Fanuc TP program (LS listing): UP021.LS

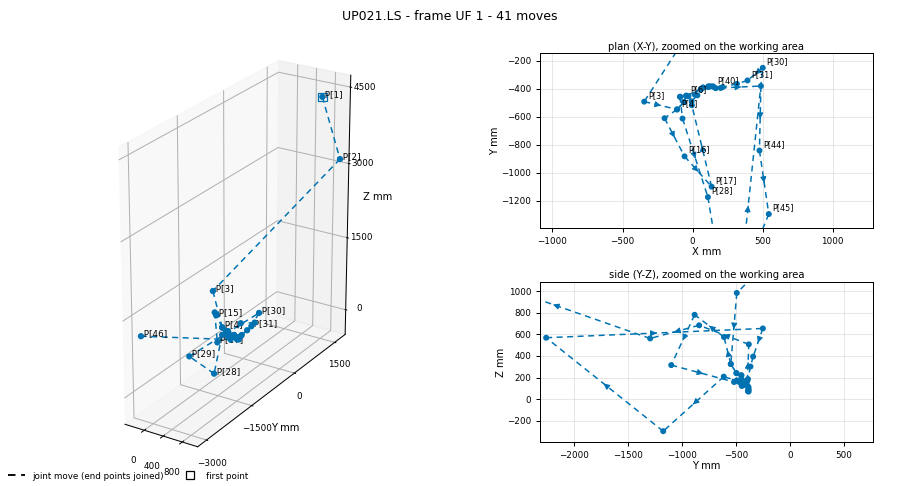
[picture p0: tool path of UP021.LS in frame UF 1, 41 of 46 moves have a stored position in this frame; points joined in program order, loops and branches not executed]
/PROG  UP021
/ATTR
OWNER		= GME;
COMMENT		= "Soldar en ST1120";
PROG_SIZE	= 17280;
CREATE		= DATE 96-06-10  TIME 20:13:44;
MODIFIED	= DATE 23-11-12  TIME 10:55:54;
FILE_NAME	= UP021;
VERSION		= 0;
LINE_COUNT	= 61;
MEMORY_SIZE	= 34620;
PROTECT		= READ_WRITE;
TCD:  STACK_SIZE	= 500,
      TASK_PRIORITY	= 50,
      TIME_SLICE	= 0,
      BUSY_LAMP_OFF	= 0,
      ABORT_REQUEST	= 0,
      PAUSE_REQUEST	= 0;
DEFAULT_GROUP	= 1,1,1,1,*;
CONTROL_CODE	= 00000000 00000000;
/APPL
/MN
   1:  UFRAME_NUM=1 ;
   2:  UTOOL_NUM=1 ;
   3:  PAYLOAD[1] ;
   4:J P[1] 100% CNT0 ACC100 TB    0.00sec,P-SPS    ;
      1:  TC_ONLINE (ON) ;
      2:  DO[23:Bloquear Rejas de Seg.]=OFF ;
      3:  TIMER[3]=RESET ;
      4:  TIMER[3]=START ;
      5:  CALL MAKRO050    ;
      6:  !Lib. de Herramientas ;
      7:  DO[80:PL>Cortina Seg.]=ON ;
      8:  DO[79:PL>1120 Herramienta]=ON ;
      9:  DO[78:Ctrl.1120 Cil.]=OFF ;
     10:  DO[77:Pos.Tomar 1120]=OFF ;
     11:  DO[76:PL>1125 Dep�sito]=ON ;
     12:  DO[74:Pos.Dejar 1125]=OFF ;
     13:  !Lib. de Anticolisiones ;
     14:  DO[41:Blq>1130R01(1)]=ON ;
     15:  DO[42:Blq>1130R01(2)]=ON ;
     16:  !Apagar Pos. Base ;
     17:  DO[15:PF0 Robot (Punto Cero)]=OFF ;
     18:  !Robot en Trayectoria ;
     19:  DO[16:SAK Robot (En camino)]=ON ;
     20:  WAIT (DI[80:Cortina Abajo] AND DI[79:1120 Soldar])    ;
     21:  DO[80:PL>Cortina Seg.]=OFF ;
     22:  DO[79:PL>1120 Herramienta]=OFF ;
     23:  WAIT (DI[23:Sin Sol.Acceso])    ;
     24:  DO[23:Bloquear Rejas de Seg.]=ON ;
     25:  TC_ONLINE (DI[80:Cortina Abajo] AND DI[79:1120 Soldar] AND M[2:Garra Vacia] AND M[30:Seg. de M�quina] AND M[31:Gpo.Suj. 1 Abierto] AND M[33:Gpo.Suj. 2 Abierto] AND M[95:Seguridad SP1] AND M[102:Seguridad SP2] AND
       :  M[103:KS2 En Reposo]) ;
       ------ ;
   5:J P[2] 100% CNT100 ACC100 TB   0.00sec,P-SPS    ;
      1:  TC_ONLINE (DI[80:Cortina Abajo] AND DI[79:1120 Soldar] AND M[2:Garra Vacia] AND M[30:Seg. de M�quina] AND M[31:Gpo.Suj. 1 Abierto] AND M[33:Gpo.Suj. 2 Abierto] AND M[95:Seguridad SP1] AND M[102:Seguridad SP2] AND
       :  M[103:KS2 En Reposo]) ;
       ------ ;
   6:J P[3] 100% CNT100 ACC100 TB   0.00sec,P-SPS    ;
      1:  TC_ONLINE (DI[80:Cortina Abajo] AND DI[79:1120 Soldar] AND M[2:Garra Vacia] AND M[30:Seg. de M�quina] AND M[31:Gpo.Suj. 1 Abierto] AND M[33:Gpo.Suj. 2 Abierto] AND M[95:Seguridad SP1] AND M[102:Seguridad SP2] AND
       :  M[103:KS2 En Reposo]) ;
       ------ ;
   7:J P[4] 100% CNT100 ACC100 TB   0.00sec,P-SPS    ;
      1:  TC_ONLINE (DI[80:Cortina Abajo] AND DI[79:1120 Soldar] AND M[2:Garra Vacia] AND M[30:Seg. de M�quina] AND M[31:Gpo.Suj. 1 Abierto] AND M[33:Gpo.Suj. 2 Abierto] AND M[95:Seguridad SP1] AND M[102:Seguridad SP2] AND
       :  M[103:KS2 En Reposo]) ;
       ------ ;
   8:J P[5] 100% CNT100 ACC100 TB   0.00sec,P-SPS    ;
      1:  TC_ONLINE (DI[80:Cortina Abajo] AND DI[79:1120 Soldar] AND M[2:Garra Vacia] AND M[30:Seg. de M�quina] AND M[31:Gpo.Suj. 1 Abierto] AND M[33:Gpo.Suj. 2 Abierto] AND M[95:Seguridad SP1] AND M[102:Seguridad SP2] AND
       :  M[103:KS2 En Reposo]) ;
       ------ ;
   9:J P[6] 100% CNT100 ACC100 TB   0.00sec,P-SPS    ;
      1:  TC_ONLINE (DI[80:Cortina Abajo] AND DI[79:1120 Soldar] AND M[2:Garra Vacia] AND M[30:Seg. de M�quina] AND M[31:Gpo.Suj. 1 Abierto] AND M[33:Gpo.Suj. 2 Abierto] AND M[95:Seguridad SP1] AND M[102:Seguridad SP2] AND
       :  M[103:KS2 En Reposo]) ;
       ------ ;
  10:J P[7] 100% CNT25 ACC100 TB   0.00sec,P-SPS    ;
      1:  TC_ONLINE (DI[80:Cortina Abajo] AND DI[79:1120 Soldar] AND M[2:Garra Vacia] AND M[30:Seg. de M�quina] AND M[31:Gpo.Suj. 1 Abierto] AND M[33:Gpo.Suj. 2 Abierto] AND M[95:Seguridad SP1] AND M[102:Seguridad SP2] AND
       :  M[103:KS2 En Reposo]) ;
       ------ ;
  11:J P[8] 100% CNT100 ACC100 TB   0.00sec,P-SPS    ;
      1:  TC_ONLINE (DI[80:Cortina Abajo] AND DI[79:1120 Soldar] AND M[2:Garra Vacia] AND M[30:Seg. de M�quina] AND M[31:Gpo.Suj. 1 Abierto] AND M[33:Gpo.Suj. 2 Abierto] AND M[95:Seguridad SP1] AND M[102:Seguridad SP2] AND
       :  M[103:KS2 En Reposo]) ;
       ------ ;
  12:  !5qa802035b_027_abps0002_L ;
  13:  !Punto de Sol. No. 10001 ;
  14:J P[9] 100% CNT0 ACC100 TB    .10sec,P-SPS Tool_Offset,PR[11] Offset,PR[12]    ;
      1:  TC_ONLINE (ON) ;
      2:  DO[23:Bloquear Rejas de Seg.]=OFF ;
      3:  WAIT (!DI[16:Paro Correcciones] AND DI[23:Sin Sol.Acceso])    ;
      4:  CALL VW_USER(Basic1,EZSP,Nr1,ProgNr=99, , ,S-Punkt=10001,Fzg_Typ=7,EIN/AUS=ON) ;
      5:  GO[2:SP1 Compensaci�n]=(R[197]) ;
      6:  WAIT (!DI[129:SZ1 Sin Fuerza] OR DI[26:Conf.Repetir])    ;
      7:  CALL MAKRO080    ;
      8:  WAIT (DI[23:Sin Sol.Acceso])    ;
      9:  DO[23:Bloquear Rejas de Seg.]=ON ;
     10:  TC_ONLINE (DI[80:Cortina Abajo] AND DI[79:1120 Soldar] AND M[2:Garra Vacia] AND M[30:Seg. de M�quina] AND M[31:Gpo.Suj. 1 Abierto] AND M[33:Gpo.Suj. 2 Abierto] AND M[95:Seguridad SP1] AND M[102:Seguridad SP2] AND
       :  M[103:KS2 En Reposo]) ;
       ------ ;
  15:J P[10] 100% CNT100 ACC100 TB   0.00sec,P-SPS    ;
      1:  TC_ONLINE (DI[80:Cortina Abajo] AND DI[79:1120 Soldar] AND M[2:Garra Vacia] AND M[30:Seg. de M�quina] AND M[31:Gpo.Suj. 1 Abierto] AND M[33:Gpo.Suj. 2 Abierto] AND M[95:Seguridad SP1] AND M[102:Seguridad SP2] AND
       :  M[103:KS2 En Reposo]) ;
       ------ ;
  16:J P[11] 100% CNT25 ACC100 TB   0.00sec,P-SPS    ;
      1:  TC_ONLINE (DI[80:Cortina Abajo] AND DI[79:1120 Soldar] AND M[2:Garra Vacia] AND M[30:Seg. de M�quina] AND M[31:Gpo.Suj. 1 Abierto] AND M[33:Gpo.Suj. 2 Abierto] AND M[95:Seguridad SP1] AND M[102:Seguridad SP2] AND
       :  M[103:KS2 En Reposo]) ;
       ------ ;
  17:J P[12] 100% CNT100 ACC100 TB   0.00sec,P-SPS    ;
      1:  TC_ONLINE (DI[80:Cortina Abajo] AND DI[79:1120 Soldar] AND M[2:Garra Vacia] AND M[30:Seg. de M�quina] AND M[31:Gpo.Suj. 1 Abierto] AND M[33:Gpo.Suj. 2 Abierto] AND M[95:Seguridad SP1] AND M[102:Seguridad SP2] AND
       :  M[103:KS2 En Reposo]) ;
       ------ ;
  18:J P[13] 100% CNT100 ACC100 TB   0.00sec,P-SPS    ;
      1:  TC_ONLINE (DI[80:Cortina Abajo] AND DI[79:1120 Soldar] AND M[2:Garra Vacia] AND M[30:Seg. de M�quina] AND M[31:Gpo.Suj. 1 Abierto] AND M[33:Gpo.Suj. 2 Abierto] AND M[95:Seguridad SP1] AND M[102:Seguridad SP2] AND
       :  M[103:KS2 En Reposo]) ;
       ------ ;
  19:J P[14] 100% CNT100 ACC100 TB   0.00sec,P-SPS    ;
      1:  TC_ONLINE (DI[80:Cortina Abajo] AND DI[79:1120 Soldar] AND M[2:Garra Vacia] AND M[30:Seg. de M�quina] AND M[31:Gpo.Suj. 1 Abierto] AND M[33:Gpo.Suj. 2 Abierto] AND M[95:Seguridad SP1] AND M[102:Seguridad SP2] AND
       :  M[103:KS2 En Reposo]) ;
       ------ ;
  20:J P[15] 100% CNT100 ACC100 TB   0.00sec,P-SPS    ;
      1:  TC_ONLINE (DI[80:Cortina Abajo] AND DI[79:1120 Soldar] AND M[2:Garra Vacia] AND M[30:Seg. de M�quina] AND M[31:Gpo.Suj. 1 Abierto] AND M[33:Gpo.Suj. 2 Abierto] AND M[95:Seguridad SP1] AND M[102:Seguridad SP2] AND
       :  M[103:KS2 En Reposo]) ;
       ------ ;
  21:J P[16] 100% CNT100 ACC100 TB   0.00sec,P-SPS    ;
      1:  TC_ONLINE (DI[80:Cortina Abajo] AND DI[79:1120 Soldar] AND M[2:Garra Vacia] AND M[30:Seg. de M�quina] AND M[31:Gpo.Suj. 1 Abierto] AND M[33:Gpo.Suj. 2 Abierto] AND M[95:Seguridad SP1] AND M[102:Seguridad SP2] AND
       :  M[103:KS2 En Reposo]) ;
       ------ ;
  22:J P[17] 100% CNT100 ACC100 TB   0.00sec,P-SPS    ;
      1:  TC_ONLINE (DI[80:Cortina Abajo] AND DI[79:1120 Soldar] AND M[2:Garra Vacia] AND M[30:Seg. de M�quina] AND M[31:Gpo.Suj. 1 Abierto] AND M[33:Gpo.Suj. 2 Abierto] AND M[95:Seguridad SP1] AND M[102:Seguridad SP2] AND
       :  M[103:KS2 En Reposo]) ;
       ------ ;
  23:J P[18] 100% CNT100 ACC100 TB   0.00sec,P-SPS    ;
      1:  TC_ONLINE (DI[80:Cortina Abajo] AND DI[79:1120 Soldar] AND M[2:Garra Vacia] AND M[30:Seg. de M�quina] AND M[31:Gpo.Suj. 1 Abierto] AND M[33:Gpo.Suj. 2 Abierto] AND M[95:Seguridad SP1] AND M[102:Seguridad SP2] AND
       :  M[103:KS2 En Reposo]) ;
       ------ ;
  24:J P[19] 100% CNT100 ACC100 TB   0.00sec,P-SPS    ;
      1:  TC_ONLINE (DI[80:Cortina Abajo] AND DI[79:1120 Soldar] AND M[2:Garra Vacia] AND M[30:Seg. de M�quina] AND M[31:Gpo.Suj. 1 Abierto] AND M[33:Gpo.Suj. 2 Abierto] AND M[95:Seguridad SP1] AND M[102:Seguridad SP2] AND
       :  M[103:KS2 En Reposo]) ;
       ------ ;
  25:  !5qa802035b_027_abps0005_L ;
  26:  !Punto de Sol. No. 10002 ;
  27:J P[20] 100% CNT0 ACC100 TB    .10sec,P-SPS Tool_Offset,PR[11] Offset,PR[12]    ;
      1:  TC_ONLINE (ON) ;
      2:  DO[23:Bloquear Rejas de Seg.]=OFF ;
      3:  WAIT (!DI[16:Paro Correcciones] AND DI[23:Sin Sol.Acceso])    ;
      4:  CALL VW_USER(Basic1,EZSP,Nr1,ProgNr=99, , ,S-Punkt=10002,Fzg_Typ=7,EIN/AUS=ON) ;
      5:  GO[2:SP1 Compensaci�n]=(R[197]+1) ;
      6:  WAIT (!DI[129:SZ1 Sin Fuerza] OR DI[26:Conf.Repetir])    ;
      7:  CALL MAKRO080    ;
      8:  WAIT (DI[23:Sin Sol.Acceso])    ;
      9:  DO[23:Bloquear Rejas de Seg.]=ON ;
     10:  TC_ONLINE (DI[80:Cortina Abajo] AND DI[79:1120 Soldar] AND M[2:Garra Vacia] AND M[30:Seg. de M�quina] AND M[31:Gpo.Suj. 1 Abierto] AND M[33:Gpo.Suj. 2 Abierto] AND M[95:Seguridad SP1] AND M[102:Seguridad SP2] AND
       :  M[103:KS2 En Reposo]) ;
       ------ ;
  28:J P[21] 100% CNT100 ACC100 TB   0.00sec,P-SPS    ;
      1:  TC_ONLINE (DI[80:Cortina Abajo] AND DI[79:1120 Soldar] AND M[2:Garra Vacia] AND M[30:Seg. de M�quina] AND M[31:Gpo.Suj. 1 Abierto] AND M[33:Gpo.Suj. 2 Abierto] AND M[95:Seguridad SP1] AND M[102:Seguridad SP2] AND
       :  M[103:KS2 En Reposo]) ;
       ------ ;
  29:J P[22] 100% CNT100 ACC100 TB   0.00sec,P-SPS    ;
      1:  TC_ONLINE (DI[80:Cortina Abajo] AND DI[79:1120 Soldar] AND M[2:Garra Vacia] AND M[30:Seg. de M�quina] AND M[31:Gpo.Suj. 1 Abierto] AND M[33:Gpo.Suj. 2 Abierto] AND M[95:Seguridad SP1] AND M[102:Seguridad SP2] AND
       :  M[103:KS2 En Reposo]) ;
       ------ ;
  30:J P[23] 100% CNT100 ACC100 TB   0.00sec,P-SPS    ;
      1:  TC_ONLINE (DI[80:Cortina Abajo] AND DI[79:1120 Soldar] AND M[2:Garra Vacia] AND M[30:Seg. de M�quina] AND M[31:Gpo.Suj. 1 Abierto] AND M[33:Gpo.Suj. 2 Abierto] AND M[95:Seguridad SP1] AND M[102:Seguridad SP2] AND
       :  M[103:KS2 En Reposo]) ;
       ------ ;
  31:J P[24] 100% CNT100 ACC100 TB   0.00sec,P-SPS    ;
      1:  TC_ONLINE (DI[80:Cortina Abajo] AND DI[79:1120 Soldar] AND M[2:Garra Vacia] AND M[30:Seg. de M�quina] AND M[31:Gpo.Suj. 1 Abierto] AND M[33:Gpo.Suj. 2 Abierto] AND M[95:Seguridad SP1] AND M[102:Seguridad SP2] AND
       :  M[103:KS2 En Reposo]) ;
       ------ ;
  32:  !5qa802035b_011_lps0009_L ;
  33:  !Punto de Sol. No. 10003 ;
  34:J P[25] 100% CNT0 ACC100 TB    .10sec,P-SPS Tool_Offset,PR[11] Offset,PR[12]    ;
      1:  TC_ONLINE (ON) ;
      2:  DO[23:Bloquear Rejas de Seg.]=OFF ;
      3:  WAIT (!DI[16:Paro Correcciones] AND DI[23:Sin Sol.Acceso])    ;
      4:  CALL VW_USER(Basic1,EZSP,Nr1,ProgNr=99, , ,S-Punkt=10003,Fzg_Typ=7,EIN/AUS=ON) ;
      5:  GO[2:SP1 Compensaci�n]=(R[197]) ;
      6:  WAIT (!DI[129:SZ1 Sin Fuerza] OR DI[26:Conf.Repetir])    ;
      7:  CALL MAKRO080    ;
      8:  WAIT (DI[23:Sin Sol.Acceso])    ;
      9:  DO[23:Bloquear Rejas de Seg.]=ON ;
     10:  TC_ONLINE (DI[80:Cortina Abajo] AND DI[79:1120 Soldar] AND M[2:Garra Vacia] AND M[30:Seg. de M�quina] AND M[31:Gpo.Suj. 1 Abierto] AND M[33:Gpo.Suj. 2 Abierto] AND M[95:Seguridad SP1] AND M[102:Seguridad SP2] AND
       :  M[103:KS2 En Reposo]) ;
       ------ ;
  35:J P[26] 100% CNT100 ACC100 TB   0.00sec,P-SPS    ;
      1:  TC_ONLINE (DI[80:Cortina Abajo] AND DI[79:1120 Soldar] AND M[2:Garra Vacia] AND M[30:Seg. de M�quina] AND M[31:Gpo.Suj. 1 Abierto] AND M[33:Gpo.Suj. 2 Abierto] AND M[95:Seguridad SP1] AND M[102:Seguridad SP2] AND
       :  M[103:KS2 En Reposo]) ;
       ------ ;
  36:J P[27] 100% CNT100 ACC100 TB   0.00sec,P-SPS    ;
      1:  TC_ONLINE (DI[80:Cortina Abajo] AND DI[79:1120 Soldar] AND M[2:Garra Vacia] AND M[30:Seg. de M�quina] AND M[31:Gpo.Suj. 1 Abierto] AND M[33:Gpo.Suj. 2 Abierto] AND M[95:Seguridad SP1] AND M[102:Seguridad SP2] AND
       :  M[103:KS2 En Reposo]) ;
       ------ ;
  37:J P[28] 100% CNT100 ACC100 TB   0.00sec,P-SPS    ;
      1:  TC_ONLINE (DI[80:Cortina Abajo] AND DI[79:1120 Soldar] AND M[2:Garra Vacia] AND M[30:Seg. de M�quina] AND M[31:Gpo.Suj. 1 Abierto] AND M[33:Gpo.Suj. 2 Abierto] AND M[95:Seguridad SP1] AND M[102:Seguridad SP2] AND
       :  M[103:KS2 En Reposo]) ;
       ------ ;
  38:J P[29] 100% CNT100 ACC100 TB   0.00sec,P-SPS    ;
      1:  TC_ONLINE (DI[80:Cortina Abajo] AND DI[79:1120 Soldar] AND M[2:Garra Vacia] AND M[30:Seg. de M�quina] AND M[31:Gpo.Suj. 1 Abierto] AND M[33:Gpo.Suj. 2 Abierto] AND M[95:Seguridad SP1] AND M[102:Seguridad SP2] AND
       :  M[103:KS2 En Reposo]) ;
       ------ ;
  39:J P[30] 100% CNT100 ACC100 TB   0.00sec,P-SPS    ;
      1:  TC_ONLINE (DI[80:Cortina Abajo] AND DI[79:1120 Soldar] AND M[2:Garra Vacia] AND M[30:Seg. de M�quina] AND M[31:Gpo.Suj. 1 Abierto] AND M[33:Gpo.Suj. 2 Abierto] AND M[95:Seguridad SP1] AND M[102:Seguridad SP2] AND
       :  M[103:KS2 En Reposo]) ;
       ------ ;
  40:J P[31] 100% CNT100 ACC100 TB   0.00sec,P-SPS    ;
      1:  TC_ONLINE (DI[80:Cortina Abajo] AND DI[79:1120 Soldar] AND M[2:Garra Vacia] AND M[30:Seg. de M�quina] AND M[31:Gpo.Suj. 1 Abierto] AND M[33:Gpo.Suj. 2 Abierto] AND M[95:Seguridad SP1] AND M[102:Seguridad SP2] AND
       :  M[103:KS2 En Reposo]) ;
       ------ ;
  41:J P[32] 100% CNT100 ACC100 TB   0.00sec,P-SPS    ;
      1:  TC_ONLINE (DI[80:Cortina Abajo] AND DI[79:1120 Soldar] AND M[2:Garra Vacia] AND M[30:Seg. de M�quina] AND M[31:Gpo.Suj. 1 Abierto] AND M[33:Gpo.Suj. 2 Abierto] AND M[95:Seguridad SP1] AND M[102:Seguridad SP2] AND
       :  M[103:KS2 En Reposo]) ;
       ------ ;
  42:J P[33] 100% CNT100 ACC100 TB   0.00sec,P-SPS    ;
      1:  TC_ONLINE (DI[80:Cortina Abajo] AND DI[79:1120 Soldar] AND M[2:Garra Vacia] AND M[30:Seg. de M�quina] AND M[31:Gpo.Suj. 1 Abierto] AND M[33:Gpo.Suj. 2 Abierto] AND M[95:Seguridad SP1] AND M[102:Seguridad SP2] AND
       :  M[103:KS2 En Reposo]) ;
       ------ ;
  43:J P[34] 100% CNT100 ACC100 TB   0.00sec,P-SPS    ;
      1:  TC_ONLINE (DI[80:Cortina Abajo] AND DI[79:1120 Soldar] AND M[2:Garra Vacia] AND M[30:Seg. de M�quina] AND M[31:Gpo.Suj. 1 Abierto] AND M[33:Gpo.Suj. 2 Abierto] AND M[95:Seguridad SP1] AND M[102:Seguridad SP2] AND
       :  M[103:KS2 En Reposo]) ;
       ------ ;
  44:J P[35] 100% CNT100 ACC100 TB   0.00sec,P-SPS    ;
      1:  TC_ONLINE (DI[80:Cortina Abajo] AND DI[79:1120 Soldar] AND M[2:Garra Vacia] AND M[30:Seg. de M�quina] AND M[31:Gpo.Suj. 1 Abierto] AND M[33:Gpo.Suj. 2 Abierto] AND M[95:Seguridad SP1] AND M[102:Seguridad SP2] AND
       :  M[103:KS2 En Reposo]) ;
       ------ ;
  45:J P[36] 100% CNT50 ACC100 TB   0.00sec,P-SPS    ;
      1:  TC_ONLINE (DI[80:Cortina Abajo] AND DI[79:1120 Soldar] AND M[2:Garra Vacia] AND M[30:Seg. de M�quina] AND M[31:Gpo.Suj. 1 Abierto] AND M[33:Gpo.Suj. 2 Abierto] AND M[95:Seguridad SP1] AND M[102:Seguridad SP2] AND
       :  M[103:KS2 En Reposo]) ;
       ------ ;
  46:  !5qa802035b_001_aps0008_L ;
  47:  !Punto de Sol. No. 10004 ;
  48:J P[37] 100% CNT0 ACC100 TB    .10sec,P-SPS Tool_Offset,PR[11] Offset,PR[12]    ;
      1:  TC_ONLINE (ON) ;
      2:  DO[23:Bloquear Rejas de Seg.]=OFF ;
      3:  WAIT (!DI[16:Paro Correcciones] AND DI[23:Sin Sol.Acceso])    ;
      4:  CALL VW_USER(Basic1,EZSP,Nr1,ProgNr=99, , ,S-Punkt=10004,Fzg_Typ=7,EIN/AUS=ON) ;
      5:  GO[2:SP1 Compensaci�n]=(R[197]) ;
      6:  WAIT (!DI[129:SZ1 Sin Fuerza] OR DI[26:Conf.Repetir])    ;
      7:  CALL MAKRO080    ;
      8:  WAIT (DI[23:Sin Sol.Acceso])    ;
      9:  DO[23:Bloquear Rejas de Seg.]=ON ;
     10:  TC_ONLINE (DI[80:Cortina Abajo] AND DI[79:1120 Soldar] AND M[2:Garra Vacia] AND M[30:Seg. de M�quina] AND M[31:Gpo.Suj. 1 Abierto] AND M[33:Gpo.Suj. 2 Abierto] AND M[95:Seguridad SP1] AND M[102:Seguridad SP2] AND
       :  M[103:KS2 En Reposo]) ;
       ------ ;
  49:J P[38] 100% CNT100 ACC100 TB   0.00sec,P-SPS    ;
      1:  TC_ONLINE (DI[80:Cortina Abajo] AND DI[79:1120 Soldar] AND M[2:Garra Vacia] AND M[30:Seg. de M�quina] AND M[31:Gpo.Suj. 1 Abierto] AND M[33:Gpo.Suj. 2 Abierto] AND M[95:Seguridad SP1] AND M[102:Seguridad SP2] AND
       :  M[103:KS2 En Reposo]) ;
       ------ ;
  50:  !5qa802035b_001_aps0001_L ;
  51:  !Punto de Sol. No. 10005 ;
  52:  !Fin de Trabajo 1 ;
  53:J P[39] 100% CNT0 ACC100 TB    0.00sec,P-SPS Tool_Offset,PR[11] Offset,PR[12]    ;
      1:  TC_ONLINE (ON) ;
      2:  DO[23:Bloquear Rejas de Seg.]=OFF ;
      3:  WAIT (!DI[16:Paro Correcciones] AND DI[23:Sin Sol.Acceso])    ;
      4:  CALL VW_USER(Basic1,EZSP,Nr1,ProgNr=99, , ,S-Punkt=10005,Fzg_Typ=7,EIN/AUS=ON) ;
      5:  GO[2:SP1 Compensaci�n]=(R[197]) ;
      6:  WAIT (!DI[129:SZ1 Sin Fuerza] OR DI[26:Conf.Repetir])    ;
      7:  CALL MAKRO080    ;
      8:  IF (!DI[145:SK1 Sin Soldadura] AND !DI[129:SZ1 Sin Fuerza]),CALL MAKRO001 ;
      9:  WAIT (DI[23:Sin Sol.Acceso])    ;
     10:  DO[23:Bloquear Rejas de Seg.]=ON ;
     11:  TC_ONLINE (DI[80:Cortina Abajo] AND DI[79:1120 Soldar] AND M[2:Garra Vacia] AND M[30:Seg. de M�quina] AND M[31:Gpo.Suj. 1 Abierto] AND M[33:Gpo.Suj. 2 Abierto] AND M[95:Seguridad SP1] AND M[102:Seguridad SP2] AND
       :  M[103:KS2 En Reposo]) ;
       ------ ;
  54:J P[40] 100% CNT100 ACC100 TB   0.00sec,P-SPS    ;
      1:  TC_ONLINE (DI[80:Cortina Abajo] AND DI[79:1120 Soldar] AND M[2:Garra Vacia] AND M[30:Seg. de M�quina] AND M[31:Gpo.Suj. 1 Abierto] AND M[33:Gpo.Suj. 2 Abierto] AND M[95:Seguridad SP1] AND M[102:Seguridad SP2] AND
       :  M[103:KS2 En Reposo]) ;
       ------ ;
  55:J P[41] 100% CNT100 ACC100 TB   0.00sec,P-SPS    ;
      1:  TC_ONLINE (DI[80:Cortina Abajo] AND DI[79:1120 Soldar] AND M[2:Garra Vacia] AND M[30:Seg. de M�quina] AND M[31:Gpo.Suj. 1 Abierto] AND M[33:Gpo.Suj. 2 Abierto] AND M[95:Seguridad SP1] AND M[102:Seguridad SP2] AND
       :  M[103:KS2 En Reposo]) ;
       ------ ;
  56:J P[42] 100% CNT100 ACC100 TB   0.00sec,P-SPS    ;
      1:  TC_ONLINE (DI[80:Cortina Abajo] AND DI[79:1120 Soldar] AND M[2:Garra Vacia] AND M[30:Seg. de M�quina] AND M[31:Gpo.Suj. 1 Abierto] AND M[33:Gpo.Suj. 2 Abierto] AND M[95:Seguridad SP1] AND M[102:Seguridad SP2] AND
       :  M[103:KS2 En Reposo]) ;
       ------ ;
  57:J P[43] 100% CNT100 ACC100 TB   0.00sec,P-SPS    ;
      1:  TC_ONLINE (ON) ;
      2:  DO[78:Ctrl.1120 Cil.]=ON ;
      3:  TC_ONLINE (DI[80:Cortina Abajo] AND M[2:Garra Vacia] AND M[30:Seg. de M�quina] AND M[31:Gpo.Suj. 1 Abierto] AND M[33:Gpo.Suj. 2 Abierto] AND M[95:Seguridad SP1] AND M[102:Seguridad SP2] AND M[103:KS2 En Reposo]) ;
       ------ ;
  58:J P[44] 100% CNT100 ACC100 TB   0.00sec,P-SPS    ;
      1:  TC_ONLINE (DI[80:Cortina Abajo] AND M[2:Garra Vacia] AND M[30:Seg. de M�quina] AND M[31:Gpo.Suj. 1 Abierto] AND M[33:Gpo.Suj. 2 Abierto] AND M[95:Seguridad SP1] AND M[102:Seguridad SP2] AND M[103:KS2 En Reposo]) ;
       ------ ;
  59:J P[45] 100% CNT100 ACC100 TB   0.00sec,P-SPS    ;
      1:  TC_ONLINE (DI[80:Cortina Abajo] AND M[2:Garra Vacia] AND M[30:Seg. de M�quina] AND M[31:Gpo.Suj. 1 Abierto] AND M[33:Gpo.Suj. 2 Abierto] AND M[95:Seguridad SP1] AND M[102:Seguridad SP2] AND M[103:KS2 En Reposo]) ;
       ------ ;
  60:  !Posicion De Salto ;
  61:J P[46] 100% CNT0 ACC100 TB    0.00sec,P-SPS    ;
      1:  TC_ONLINE (ON) ;
      2:  DO[23:Bloquear Rejas de Seg.]=OFF ;
      3:  TIMER[3]=STOP ;
      4:  WAIT (DI[23:Sin Sol.Acceso])    ;
      5:  DO[23:Bloquear Rejas de Seg.]=ON ;
      6:  TC_ONLINE (DI[80:Cortina Abajo] AND M[2:Garra Vacia] AND M[30:Seg. de M�quina] AND M[31:Gpo.Suj. 1 Abierto] AND M[33:Gpo.Suj. 2 Abierto] AND M[95:Seguridad SP1] AND M[102:Seguridad SP2] AND M[103:KS2 En Reposo]) ;
       ------ ;
/POS
P[1]{
   GP1:
	UF : 1, UT : 1,		CONFIG : 'N U T, 0, 0, 0',
	X =   950.692  mm,	Y =  1172.599  mm,	Z =  4505.112  mm,
	W =   -48.429 deg,	P =    23.656 deg,	R =    42.815 deg
   GP2:
	UF : 1, UT : 1,
	J1=   100.000  mm
   GP3:
	UF : 1, UT : 1,
	J1=   100.000  mm
   GP4:
	UF : 1, UT : 1,
	J1=     0.000  mm
};
P[2]{
   GP1:
	UF : 1, UT : 1,		CONFIG : 'N U T, 0, 0, 0',
	X =  1054.409  mm,	Y =  1681.744  mm,	Z =  3150.066  mm,
	W =   -40.639 deg,	P =    51.707 deg,	R =    52.972 deg
   GP2:
	UF : 1, UT : 1,
	J1=   218.351  mm
   GP3:
	UF : 1, UT : 1,
	J1=   101.068  mm
   GP4:
	UF : 1, UT : 1,
	J1=     0.000  mm
};
P[3]{
   GP1:
	UF : 1, UT : 1,		CONFIG : 'N U T, 0, 0, 0',
	X =  -344.966  mm,	Y =  -490.858  mm,	Z =   983.696  mm,
	W =   158.707 deg,	P =    22.388 deg,	R =   120.572 deg
   GP2:
	UF : 1, UT : 1,
	J1=   224.600  mm
   GP3:
	UF : 1, UT : 1,
	J1=   100.000  mm
   GP4:
	UF : 1, UT : 1,
	J1=     0.000  mm
};
P[4]{
   GP1:
	UF : 1, UT : 1,		CONFIG : 'N U T, 0, 0, 0',
	X =  -110.484  mm,	Y =  -546.469  mm,	Z =   324.761  mm,
	W =   128.459 deg,	P =      .252 deg,	R =   104.513 deg
   GP2:
	UF : 1, UT : 1,
	J1=   224.600  mm
   GP3:
	UF : 1, UT : 1,
	J1=   100.000  mm
   GP4:
	UF : 1, UT : 1,
	J1=     0.000  mm
};
P[5]{
   GP1:
	UF : 1, UT : 1,		CONFIG : 'N U T, 0, 0, 0',
	X =   -61.595  mm,	Y =  -494.149  mm,	Z =   240.455  mm,
	W =   137.290 deg,	P =    10.643 deg,	R =    98.484 deg
   GP2:
	UF : 1, UT : 1,
	J1=   211.334  mm
   GP3:
	UF : 1, UT : 1,
	J1=   100.000  mm
   GP4:
	UF : 1, UT : 1,
	J1=     0.000  mm
};
P[6]{
   GP1:
	UF : 1, UT : 1,		CONFIG : 'N U T, 0, 0, 0',
	X =   -44.806  mm,	Y =  -448.350  mm,	Z =   220.014  mm,
	W =   135.855 deg,	P =      .253 deg,	R =   104.512 deg
   GP2:
	UF : 1, UT : 1,
	J1=   184.118  mm
   GP3:
	UF : 1, UT : 1,
	J1=   100.000  mm
   GP4:
	UF : 1, UT : 1,
	J1=     0.000  mm
};
P[7]{
   GP1:
	UF : 1, UT : 1,		CONFIG : 'N U T, 0, 0, 0',
	X =    58.909  mm,	Y =  -401.090  mm,	Z =   152.594  mm,
	W =   129.648 deg,	P =      .253 deg,	R =   104.512 deg
   GP2:
	UF : 1, UT : 1,
	J1=   118.200  mm
   GP3:
	UF : 1, UT : 1,
	J1=   100.000  mm
   GP4:
	UF : 1, UT : 1,
	J1=     0.000  mm
};
P[8]{
   GP1:
	UF : 1, UT : 1,		CONFIG : 'N U T, 0, 0, 0',
	X =    75.171  mm,	Y =  -390.661  mm,	Z =   119.968  mm,
	W =   137.632 deg,	P =      .254 deg,	R =   104.511 deg
   GP2:
	UF : 1, UT : 1,
	J1=   101.000  mm
   GP3:
	UF : 1, UT : 1,
	J1=   100.000  mm
   GP4:
	UF : 1, UT : 1,
	J1=     0.000  mm
};
P[9]{
   GP1:
	UF : 1, UT : 1,		CONFIG : 'N U T, 0, 0, 0',
	X =    82.910  mm,	Y =  -389.957  mm,	Z =   122.320  mm,
	W =   131.445 deg,	P =     2.600 deg,	R =   102.831 deg
   GP2:
	UF : 1, UT : 1,
	J1=    26.100  mm
   GP3:
	UF : 1, UT : 1,
	J1=   106.000  mm
   GP4:
	UF : 1, UT : 1,
	J1=     0.000  mm
};
P[10]{
   GP1:
	UF : 1, UT : 1,		CONFIG : 'N U T, 0, 0, 0',
	X =    75.034  mm,	Y =  -390.135  mm,	Z =   119.965  mm,
	W =   137.632 deg,	P =      .254 deg,	R =   104.511 deg
   GP2:
	UF : 1, UT : 1,
	J1=   102.900  mm
   GP3:
	UF : 1, UT : 1,
	J1=   100.000  mm
   GP4:
	UF : 1, UT : 1,
	J1=     0.000  mm
};
P[11]{
   GP1:
	UF : 1, UT : 1,		CONFIG : 'N U T, 0, 0, 0',
	X =    59.654  mm,	Y =  -403.980  mm,	Z =   152.604  mm,
	W =   129.652 deg,	P =     -.774 deg,	R =   103.660 deg
   GP2:
	UF : 1, UT : 1,
	J1=   136.200  mm
   GP3:
	UF : 1, UT : 1,
	J1=   100.000  mm
   GP4:
	UF : 1, UT : 1,
	J1=     0.000  mm
};
P[12]{
   GP1:
	UF : 1, UT : 1,		CONFIG : 'N U T, 0, 0, 0',
	X =   -44.805  mm,	Y =  -448.350  mm,	Z =   220.014  mm,
	W =   135.855 deg,	P =      .253 deg,	R =   104.512 deg
   GP2:
	UF : 1, UT : 1,
	J1=   184.118  mm
   GP3:
	UF : 1, UT : 1,
	J1=   100.000  mm
   GP4:
	UF : 1, UT : 1,
	J1=     0.000  mm
};
P[13]{
   GP1:
	UF : 1, UT : 1,		CONFIG : 'N U T, 0, 0, 0',
	X =   -61.595  mm,	Y =  -494.149  mm,	Z =   240.455  mm,
	W =   137.290 deg,	P =    10.643 deg,	R =    98.484 deg
   GP2:
	UF : 1, UT : 1,
	J1=   211.334  mm
   GP3:
	UF : 1, UT : 1,
	J1=   100.000  mm
   GP4:
	UF : 1, UT : 1,
	J1=     0.000  mm
};
P[14]{
   GP1:
	UF : 1, UT : 1,		CONFIG : 'N U T, 0, 0, 0',
	X =  -110.484  mm,	Y =  -546.469  mm,	Z =   324.761  mm,
	W =   128.459 deg,	P =      .252 deg,	R =   104.513 deg
   GP2:
	UF : 1, UT : 1,
	J1=   211.334  mm
   GP3:
	UF : 1, UT : 1,
	J1=   100.000  mm
   GP4:
	UF : 1, UT : 1,
	J1=     0.000  mm
};
P[15]{
   GP1:
	UF : 1, UT : 1,		CONFIG : 'N U T, 0, 0, 0',
	X =  -199.651  mm,	Y =  -609.213  mm,	Z =   574.533  mm,
	W =   124.434 deg,	P =      .251 deg,	R =   104.513 deg
   GP2:
	UF : 1, UT : 1,
	J1=   100.000  mm
   GP3:
	UF : 1, UT : 1,
	J1=   100.000  mm
   GP4:
	UF : 1, UT : 1,
	J1=     0.000  mm
};
P[16]{
   GP1:
	UF : 1, UT : 1,		CONFIG : 'N U T, 0, 0, 0',
	X =   -56.867  mm,	Y =  -881.581  mm,	Z =   781.234  mm,
	W =   118.667 deg,	P =    17.320 deg,	R =   107.993 deg
   GP2:
	UF : 1, UT : 1,
	J1=   174.542  mm
   GP3:
	UF : 1, UT : 1,
	J1=   100.000  mm
   GP4:
	UF : 1, UT : 1,
	J1=     0.000  mm
};
P[17]{
   GP1:
	UF : 1, UT : 1,		CONFIG : 'N U T, 0, 0, 0',
	X =   136.281  mm,	Y = -1098.211  mm,	Z =   314.949  mm,
	W =   125.715 deg,	P =    34.265 deg,	R =   148.281 deg
   GP2:
	UF : 1, UT : 1,
	J1=   100.000  mm
   GP3:
	UF : 1, UT : 1,
	J1=   100.000  mm
   GP4:
	UF : 1, UT : 1,
	J1=     0.000  mm
};
P[18]{
   GP1:
	UF : 1, UT : 1,		CONFIG : 'N U T, 0, 0, 0',
	X =    -4.846  mm,	Y =  -516.273  mm,	Z =   158.480  mm,
	W =   132.906 deg,	P =    55.857 deg,	R =   179.278 deg
   GP2:
	UF : 1, UT : 1,
	J1=   100.000  mm
   GP3:
	UF : 1, UT : 1,
	J1=   100.000  mm
   GP4:
	UF : 1, UT : 1,
	J1=     0.000  mm
};
P[19]{
   GP1:
	UF : 1, UT : 1,		CONFIG : 'N U T, 0, 0, 0',
	X =    15.636  mm,	Y =  -440.136  mm,	Z =   123.655  mm,
	W =   132.904 deg,	P =    55.857 deg,	R =   179.276 deg
   GP2:
	UF : 1, UT : 1,
	J1=   127.700  mm
   GP3:
	UF : 1, UT : 1,
	J1=   100.900  mm
   GP4:
	UF : 1, UT : 1,
	J1=     0.000  mm
};
P[20]{
   GP1:
	UF : 1, UT : 1,		CONFIG : 'N U T, 0, 0, 0',
	X =    62.278  mm,	Y =  -412.987  mm,	Z =    84.609  mm,
	W =   132.888 deg,	P =    55.854 deg,	R =   179.256 deg
   GP2:
	UF : 1, UT : 1,
	J1=    30.000  mm
   GP3:
	UF : 1, UT : 1,
	J1=   104.100  mm
   GP4:
	UF : 1, UT : 1,
	J1=     0.000  mm
};
P[21]{
   GP1:
	UF : 1, UT : 1,		CONFIG : 'N U T, 0, 0, 0',
	X =    34.437  mm,	Y =  -445.741  mm,	Z =   122.986  mm,
	W =   145.778 deg,	P =    65.405 deg,	R =  -168.189 deg
   GP2:
	UF : 1, UT : 1,
	J1=   125.600  mm
   GP3:
	UF : 1, UT : 1,
	J1=   100.000  mm
   GP4:
	UF : 1, UT : 1,
	J1=     0.000  mm
};
P[22]{
   GP1:
	UF : 1, UT : 1,		CONFIG : 'N U T, 0, 0, 0',
	X =    -6.262  mm,	Y =  -488.570  mm,	Z =   174.232  mm,
	W =   116.754 deg,	P =    65.404 deg,	R =  -168.183 deg
   GP2:
	UF : 1, UT : 1,
	J1=   120.000  mm
   GP3:
	UF : 1, UT : 1,
	J1=   100.000  mm
   GP4:
	UF : 1, UT : 1,
	J1=     0.000  mm
};
P[23]{
   GP1:
	UF : 1, UT : 1,		CONFIG : 'N U T, 0, 0, 0',
	X =   -29.399  mm,	Y =  -453.127  mm,	Z =   164.016  mm,
	W =   107.763 deg,	P =    80.231 deg,	R =   174.413 deg
   GP2:
	UF : 1, UT : 1,
	J1=   101.176  mm
   GP3:
	UF : 1, UT : 1,
	J1=   100.000  mm
   GP4:
	UF : 1, UT : 1,
	J1=     0.000  mm
};
P[24]{
   GP1:
	UF : 1, UT : 1,		CONFIG : 'N U T, 0, 0, 0',
	X =   -87.311  mm,	Y =  -456.206  mm,	Z =   173.888  mm,
	W =    81.493 deg,	P =    80.230 deg,	R =   174.412 deg
   GP2:
	UF : 1, UT : 1,
	J1=   101.176  mm
   GP3:
	UF : 1, UT : 1,
	J1=   100.000  mm
   GP4:
	UF : 1, UT : 1,
	J1=     0.000  mm
};
P[25]{
   GP1:
	UF : 1, UT : 1,		CONFIG : 'N U T, 0, 0, 0',
	X =   -90.166  mm,	Y =  -454.736  mm,	Z =   151.432  mm,
	W =    81.076 deg,	P =    81.576 deg,	R =   173.993 deg
   GP2:
	UF : 1, UT : 1,
	J1=    18.200  mm
   GP3:
	UF : 1, UT : 1,
	J1=   100.000  mm
   GP4:
	UF : 1, UT : 1,
	J1=     0.000  mm
};
P[26]{
   GP1:
	UF : 1, UT : 1,		CONFIG : 'N U T, 0, 0, 0',
	X =   -89.795  mm,	Y =  -455.968  mm,	Z =   159.374  mm,
	W =    81.494 deg,	P =    80.230 deg,	R =   174.413 deg
   GP2:
	UF : 1, UT : 1,
	J1=    60.000  mm
   GP3:
	UF : 1, UT : 1,
	J1=   100.000  mm
   GP4:
	UF : 1, UT : 1,
	J1=     0.000  mm
};
P[27]{
   GP1:
	UF : 1, UT : 1,		CONFIG : 'N U T, 0, 0, 0',
	X =   -71.408  mm,	Y =  -611.623  mm,	Z =   208.103  mm,
	W =   148.355 deg,	P =    78.725 deg,	R =  -117.120 deg
   GP2:
	UF : 1, UT : 1,
	J1=    97.500  mm
   GP3:
	UF : 1, UT : 1,
	J1=   100.000  mm
   GP4:
	UF : 1, UT : 1,
	J1=     0.000  mm
};
P[28]{
   GP1:
	UF : 1, UT : 1,		CONFIG : 'N U T, 0, 0, 0',
	X =   109.801  mm,	Y = -1172.579  mm,	Z =  -297.416  mm,
	W =   179.066 deg,	P =    51.056 deg,	R =   -84.575 deg
   GP2:
	UF : 1, UT : 1,
	J1=   100.000  mm
   GP3:
	UF : 1, UT : 1,
	J1=   100.000  mm
   GP4:
	UF : 1, UT : 1,
	J1=     0.000  mm
};
P[29]{
   GP1:
	UF : 1, UT : 1,		CONFIG : 'N U T, 0, 0, -1',
	X =   289.573  mm,	Y = -2257.289  mm,	Z =   568.711  mm,
	W =   152.860 deg,	P =    76.851 deg,	R =    32.992 deg
   GP2:
	UF : 1, UT : 1,
	J1=   100.000  mm
   GP3:
	UF : 1, UT : 1,
	J1=   100.000  mm
   GP4:
	UF : 1, UT : 1,
	J1=     0.000  mm
};
P[30]{
   GP1:
	UF : 1, UT : 1,		CONFIG : 'N U T, 0, 0, -1',
	X =   501.660  mm,	Y =  -249.278  mm,	Z =   654.602  mm,
	W =  -157.291 deg,	P =    13.937 deg,	R =    86.449 deg
   GP2:
	UF : 1, UT : 1,
	J1=   100.000  mm
   GP3:
	UF : 1, UT : 1,
	J1=   100.000  mm
   GP4:
	UF : 1, UT : 1,
	J1=     0.000  mm
};
P[31]{
   GP1:
	UF : 1, UT : 1,		CONFIG : 'N U T, 0, 0, -1',
	X =   392.772  mm,	Y =  -339.449  mm,	Z =   393.993  mm,
	W =  -143.269 deg,	P =     2.576 deg,	R =    95.382 deg
   GP2:
	UF : 1, UT : 1,
	J1=   100.000  mm
   GP3:
	UF : 1, UT : 1,
	J1=   100.000  mm
   GP4:
	UF : 1, UT : 1,
	J1=     0.000  mm
};
P[32]{
   GP1:
	UF : 1, UT : 1,		CONFIG : 'N U T, 0, 0, -1',
	X =   317.084  mm,	Y =  -363.754  mm,	Z =   301.558  mm,
	W =  -138.857 deg,	P =      .698 deg,	R =    93.660 deg
   GP2:
	UF : 1, UT : 1,
	J1=   100.000  mm
   GP3:
	UF : 1, UT : 1,
	J1=   100.000  mm
   GP4:
	UF : 1, UT : 1,
	J1=     0.000  mm
};
P[33]{
   GP1:
	UF : 1, UT : 1,		CONFIG : 'N U T, 0, 0, -1',
	X =   213.898  mm,	Y =  -387.486  mm,	Z =   186.233  mm,
	W =  -138.756 deg,	P =    -4.371 deg,	R =    89.310 deg
   GP2:
	UF : 1, UT : 1,
	J1=    95.000  mm
   GP3:
	UF : 1, UT : 1,
	J1=   100.000  mm
   GP4:
	UF : 1, UT : 1,
	J1=     0.000  mm
};
P[34]{
   GP1:
	UF : 1, UT : 1,		CONFIG : 'N U T, 0, 0, -1',
	X =   145.922  mm,	Y =  -381.717  mm,	Z =   108.781  mm,
	W =  -138.706 deg,	P =    -5.062 deg,	R =    88.701 deg
   GP2:
	UF : 1, UT : 1,
	J1=    80.923  mm
   GP3:
	UF : 1, UT : 1,
	J1=   100.000  mm
   GP4:
	UF : 1, UT : 1,
	J1=     0.000  mm
};
P[35]{
   GP1:
	UF : 1, UT : 1,		CONFIG : 'N U T, 0, 0, -1',
	X =   128.081  mm,	Y =  -381.091  mm,	Z =    88.382  mm,
	W =  -138.895 deg,	P =      .962 deg,	R =    93.972 deg
   GP2:
	UF : 1, UT : 1,
	J1=    69.269  mm
   GP3:
	UF : 1, UT : 1,
	J1=   100.000  mm
   GP4:
	UF : 1, UT : 1,
	J1=     0.000  mm
};
P[36]{
   GP1:
	UF : 1, UT : 1,		CONFIG : 'N U T, 0, 0, -1',
	X =   113.237  mm,	Y =  -381.295  mm,	Z =    70.308  mm,
	W =  -138.880 deg,	P =     1.734 deg,	R =    94.646 deg
   GP2:
	UF : 1, UT : 1,
	J1=    67.700  mm
   GP3:
	UF : 1, UT : 1,
	J1=   100.000  mm
   GP4:
	UF : 1, UT : 1,
	J1=     0.000  mm
};
P[37]{
   GP1:
	UF : 1, UT : 1,		CONFIG : 'N U T, 0, 0, -1',
	X =   107.322  mm,	Y =  -384.511  mm,	Z =    77.121  mm,
	W =  -138.633 deg,	P =     5.935 deg,	R =    98.336 deg
   GP2:
	UF : 1, UT : 1,
	J1=    17.300  mm
   GP3:
	UF : 1, UT : 1,
	J1=   100.000  mm
   GP4:
	UF : 1, UT : 1,
	J1=     0.000  mm
};
P[38]{
   GP1:
	UF : 1, UT : 1,		CONFIG : 'N U T, 0, 0, -1',
	X =   111.696  mm,	Y =  -387.281  mm,	Z =    72.431  mm,
	W =  -141.632 deg,	P =     5.935 deg,	R =    98.336 deg
   GP2:
	UF : 1, UT : 1,
	J1=    50.000  mm
   GP3:
	UF : 1, UT : 1,
	J1=   100.000  mm
   GP4:
	UF : 1, UT : 1,
	J1=     0.000  mm
};
P[39]{
   GP1:
	UF : 1, UT : 1,		CONFIG : 'N U T, 0, 0, -1',
	X =   142.519  mm,	Y =  -380.214  mm,	Z =    79.698  mm,
	W =  -142.343 deg,	P =     7.352 deg,	R =    97.024 deg
   GP2:
	UF : 1, UT : 1,
	J1=    16.100  mm
   GP3:
	UF : 1, UT : 1,
	J1=   103.800  mm
   GP4:
	UF : 1, UT : 1,
	J1=     0.000  mm
};
P[40]{
   GP1:
	UF : 1, UT : 1,		CONFIG : 'N U T, 0, 0, -1',
	X =   148.718  mm,	Y =  -384.677  mm,	Z =    77.305  mm,
	W =  -144.274 deg,	P =      .613 deg,	R =    92.302 deg
   GP2:
	UF : 1, UT : 1,
	J1=    85.100  mm
   GP3:
	UF : 1, UT : 1,
	J1=   100.000  mm
   GP4:
	UF : 1, UT : 1,
	J1=     0.000  mm
};
P[41]{
   GP1:
	UF : 1, UT : 1,		CONFIG : 'N U T, 0, 0, -1',
	X =   165.830  mm,	Y =  -395.018  mm,	Z =   120.892  mm,
	W =  -144.199 deg,	P =    -3.494 deg,	R =    89.343 deg
   GP2:
	UF : 1, UT : 1,
	J1=   116.574  mm
   GP3:
	UF : 1, UT : 1,
	J1=   100.000  mm
   GP4:
	UF : 1, UT : 1,
	J1=     0.000  mm
};
P[42]{
   GP1:
	UF : 1, UT : 1,		CONFIG : 'N U T, 0, 0, -1',
	X =   201.075  mm,	Y =  -393.061  mm,	Z =   169.981  mm,
	W =  -144.274 deg,	P =      .613 deg,	R =    92.302 deg
   GP2:
	UF : 1, UT : 1,
	J1=   101.152  mm
   GP3:
	UF : 1, UT : 1,
	J1=   100.000  mm
   GP4:
	UF : 1, UT : 1,
	J1=     0.000  mm
};
P[43]{
   GP1:
	UF : 1, UT : 1,		CONFIG : 'N U T, 0, 0, -1',
	X =   488.372  mm,	Y =  -379.456  mm,	Z =   507.436  mm,
	W =  -166.646 deg,	P =    27.151 deg,	R =    80.219 deg
   GP2:
	UF : 1, UT : 1,
	J1=   150.000  mm
   GP3:
	UF : 1, UT : 1,
	J1=   100.000  mm
   GP4:
	UF : 1, UT : 1,
	J1=     0.000  mm
};
P[44]{
   GP1:
	UF : 1, UT : 1,		CONFIG : 'N U T, 0, 0, -1',
	X =   477.930  mm,	Y =  -840.093  mm,	Z =   683.771  mm,
	W =  -170.668 deg,	P =    36.461 deg,	R =    74.576 deg
   GP2:
	UF : 1, UT : 1,
	J1=   100.000  mm
   GP3:
	UF : 1, UT : 1,
	J1=   100.000  mm
   GP4:
	UF : 1, UT : 1,
	J1=     0.000  mm
};
P[45]{
   GP1:
	UF : 1, UT : 1,		CONFIG : 'N U T, 0, 0, -1',
	X =   544.722  mm,	Y = -1293.835  mm,	Z =   562.077  mm,
	W =  -165.196 deg,	P =    45.233 deg,	R =   102.557 deg
   GP2:
	UF : 1, UT : 1,
	J1=   100.000  mm
   GP3:
	UF : 1, UT : 1,
	J1=   100.000  mm
   GP4:
	UF : 1, UT : 1,
	J1=     0.000  mm
};
P[46]{
   GP1:
	UF : 1, UT : 1,		CONFIG : 'N U T, 0, 0, 0',
	X =  -184.141  mm,	Y = -3059.016  mm,	Z =  1178.475  mm,
	W =     1.989 deg,	P =    75.979 deg,	R =   -87.030 deg
   GP2:
	UF : 1, UT : 1,
	J1=   100.000  mm
   GP3:
	UF : 1, UT : 1,
	J1=   100.000  mm
   GP4:
	UF : 1, UT : 1,
	J1=     0.000  mm
};
/END
